// TIA Portal V19 export
TYPE "_IOL_VmData"
   STRUCT
      ValveCycles : DInt;   // Valve Cycles since reset
      OpeningTime : Int;   // milliseconds
      ClosingTime : Int;   // milliseconds
      ObjErrorTime : Int;   // milliseconds
      spare : Array[1..30] of Byte;   // For Future Use
   END_STRUCT;
END_TYPE
